{attribute 'qualified_only'}
TYPE E_MMTrafficLightColor :
(
	eMMTrafficLightColor_NA		:= -1,
	eMMTrafficLightColor_Green	:= 0,
	eMMTrafficLightColor_Red	:= 1
);
END_TYPE
//  eMMTrafficLightColor_NA = '-1'

(* stored: Version 1.1.0.1, ProductVersion 3.1.4024.5
   EnumerationTextList E_MMTrafficLightColor: Id {afb261f9-7f48-49cd-b5e1-e67dd0f380f5} *)
